// TIA Portal V19 export
FUNCTION "Area03_ITF" : Void   // FC22, LAD
// stored: SetENOAutomatically false
BEGIN

REGION Network 2: AREA ITF
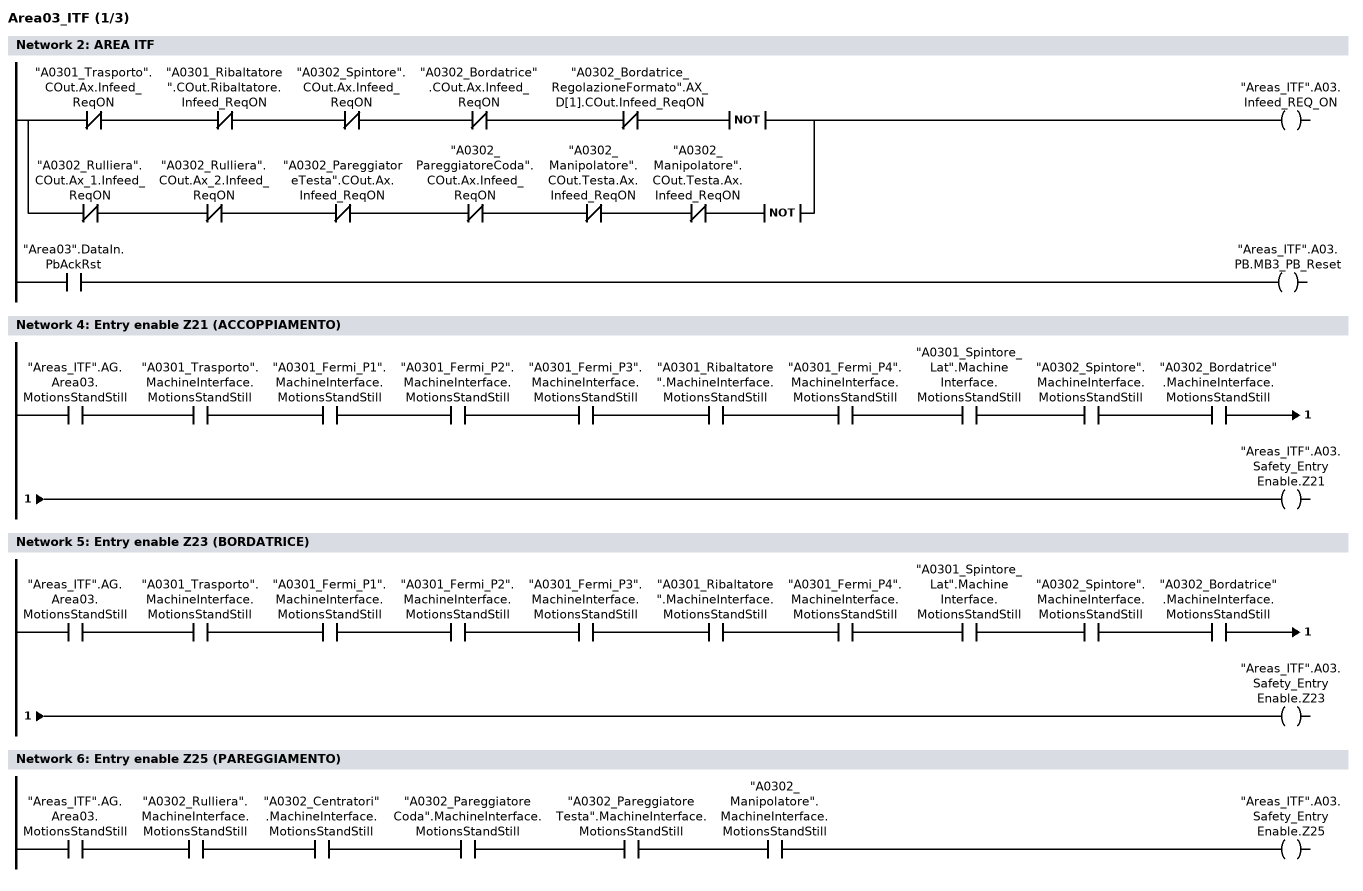
   RUNG wire#powerrail
      I_Contact( "A0301_Trasporto".COut.Ax.Infeed_ReqON )
      I_Contact( "A0301_Ribaltatore".COut.Ribaltatore.Infeed_ReqON )
      I_Contact( "A0302_Spintore".COut.Ax.Infeed_ReqON )
      I_Contact( "A0302_Bordatrice".COut.Ax.Infeed_ReqON )
      I_Contact( "A0302_Bordatrice_RegolazioneFormato".AX_D[1].COut.Infeed_ReqON )
      Not()
      wire#w1
      Coil( "Areas_ITF".A03.Infeed_REQ_ON )
   END_RUNG
   RUNG wire#powerrail
      I_Contact( "A0302_Rulliera".COut.Ax_1.Infeed_ReqON )
      I_Contact( "A0302_Rulliera".COut.Ax_2.Infeed_ReqON )
      I_Contact( "A0302_PareggiatoreTesta".COut.Ax.Infeed_ReqON )
      I_Contact( "A0302_PareggiatoreCoda".COut.Ax.Infeed_ReqON )
      I_Contact( "A0302_Manipolatore".COut.Testa.Ax.Infeed_ReqON )
      I_Contact( "A0302_Manipolatore".COut.Testa.Ax.Infeed_ReqON )
      Not()
   END_RUNG wire#w1
   RUNG wire#powerrail
      Contact( "Area03".DataIn.PbAckRst )
      Coil( "Areas_ITF".A03.PB.MB3_PB_Reset )
   END_RUNG
   // the same network as SCL:
   "Areas_ITF".A03.Infeed_REQ_ON := NOT (NOT "A0301_Trasporto".COut.Ax.Infeed_ReqON AND NOT "A0301_Ribaltatore".COut.Ribaltatore.Infeed_ReqON AND NOT "A0302_Spintore".COut.Ax.Infeed_ReqON AND NOT "A0302_Bordatrice".COut.Ax.Infeed_ReqON AND NOT "A0302_Bordatrice_RegolazioneFormato".AX_D[1].COut.Infeed_ReqON) OR NOT (NOT "A0302_Rulliera".COut.Ax_1.Infeed_ReqON AND NOT "A0302_Rulliera".COut.Ax_2.Infeed_ReqON AND NOT "A0302_PareggiatoreTesta".COut.Ax.Infeed_ReqON AND NOT "A0302_PareggiatoreCoda".COut.Ax.Infeed_ReqON AND NOT "A0302_Manipolatore".COut.Testa.Ax.Infeed_ReqON AND NOT "A0302_Manipolatore".COut.Testa.Ax.Infeed_ReqON);
   "Areas_ITF".A03.PB.MB3_PB_Reset := "Area03".DataIn.PbAckRst;
END_REGION

REGION Network 3: >
END_REGION

REGION Network 4: Entry enable Z21 (ACCOPPIAMENTO)
   RUNG wire#powerrail
      Contact( "Areas_ITF".AG.Area03.MotionsStandStill )
      Contact( "A0301_Trasporto".MachineInterface.MotionsStandStill )
      Contact( "A0301_Fermi_P1".MachineInterface.MotionsStandStill )
      Contact( "A0301_Fermi_P2".MachineInterface.MotionsStandStill )
      Contact( "A0301_Fermi_P3".MachineInterface.MotionsStandStill )
      Contact( "A0301_Ribaltatore".MachineInterface.MotionsStandStill )
      Contact( "A0301_Fermi_P4".MachineInterface.MotionsStandStill )
      Contact( "A0301_Spintore_Lat".MachineInterface.MotionsStandStill )
      Contact( "A0302_Spintore".MachineInterface.MotionsStandStill )
      Contact( "A0302_Bordatrice".MachineInterface.MotionsStandStill )
      Coil( "Areas_ITF".A03.Safety_EntryEnable.Z21 )
   END_RUNG
   // the same network as SCL:
   "Areas_ITF".A03.Safety_EntryEnable.Z21 := "Areas_ITF".AG.Area03.MotionsStandStill AND "A0301_Trasporto".MachineInterface.MotionsStandStill AND "A0301_Fermi_P1".MachineInterface.MotionsStandStill AND "A0301_Fermi_P2".MachineInterface.MotionsStandStill AND "A0301_Fermi_P3".MachineInterface.MotionsStandStill AND "A0301_Ribaltatore".MachineInterface.MotionsStandStill AND "A0301_Fermi_P4".MachineInterface.MotionsStandStill AND "A0301_Spintore_Lat".MachineInterface.MotionsStandStill AND "A0302_Spintore".MachineInterface.MotionsStandStill AND "A0302_Bordatrice".MachineInterface.MotionsStandStill;
END_REGION

REGION Network 5: Entry enable Z23 (BORDATRICE)
   RUNG wire#powerrail
      Contact( "Areas_ITF".AG.Area03.MotionsStandStill )
      Contact( "A0301_Trasporto".MachineInterface.MotionsStandStill )
      Contact( "A0301_Fermi_P1".MachineInterface.MotionsStandStill )
      Contact( "A0301_Fermi_P2".MachineInterface.MotionsStandStill )
      Contact( "A0301_Fermi_P3".MachineInterface.MotionsStandStill )
      Contact( "A0301_Ribaltatore".MachineInterface.MotionsStandStill )
      Contact( "A0301_Fermi_P4".MachineInterface.MotionsStandStill )
      Contact( "A0301_Spintore_Lat".MachineInterface.MotionsStandStill )
      Contact( "A0302_Spintore".MachineInterface.MotionsStandStill )
      Contact( "A0302_Bordatrice".MachineInterface.MotionsStandStill )
      Coil( "Areas_ITF".A03.Safety_EntryEnable.Z23 )
   END_RUNG
   // the same network as SCL:
   "Areas_ITF".A03.Safety_EntryEnable.Z23 := "Areas_ITF".AG.Area03.MotionsStandStill AND "A0301_Trasporto".MachineInterface.MotionsStandStill AND "A0301_Fermi_P1".MachineInterface.MotionsStandStill AND "A0301_Fermi_P2".MachineInterface.MotionsStandStill AND "A0301_Fermi_P3".MachineInterface.MotionsStandStill AND "A0301_Ribaltatore".MachineInterface.MotionsStandStill AND "A0301_Fermi_P4".MachineInterface.MotionsStandStill AND "A0301_Spintore_Lat".MachineInterface.MotionsStandStill AND "A0302_Spintore".MachineInterface.MotionsStandStill AND "A0302_Bordatrice".MachineInterface.MotionsStandStill;
END_REGION

REGION Network 6: Entry enable Z25 (PAREGGIAMENTO)
   RUNG wire#powerrail
      Contact( "Areas_ITF".AG.Area03.MotionsStandStill )
      Contact( "A0302_Rulliera".MachineInterface.MotionsStandStill )
      Contact( "A0302_Centratori".MachineInterface.MotionsStandStill )
      Contact( "A0302_PareggiatoreCoda".MachineInterface.MotionsStandStill )
      Contact( "A0302_PareggiatoreTesta".MachineInterface.MotionsStandStill )
      Contact( "A0302_Manipolatore".MachineInterface.MotionsStandStill )
      Coil( "Areas_ITF".A03.Safety_EntryEnable.Z25 )
   END_RUNG
   // the same network as SCL:
   "Areas_ITF".A03.Safety_EntryEnable.Z25 := "Areas_ITF".AG.Area03.MotionsStandStill AND "A0302_Rulliera".MachineInterface.MotionsStandStill AND "A0302_Centratori".MachineInterface.MotionsStandStill AND "A0302_PareggiatoreCoda".MachineInterface.MotionsStandStill AND "A0302_PareggiatoreTesta".MachineInterface.MotionsStandStill AND "A0302_Manipolatore".MachineInterface.MotionsStandStill;
END_REGION

REGION Network 7: < < < < CTRL SAFE > > > >
END_REGION

REGION Network 8: Ctrl Safe S120
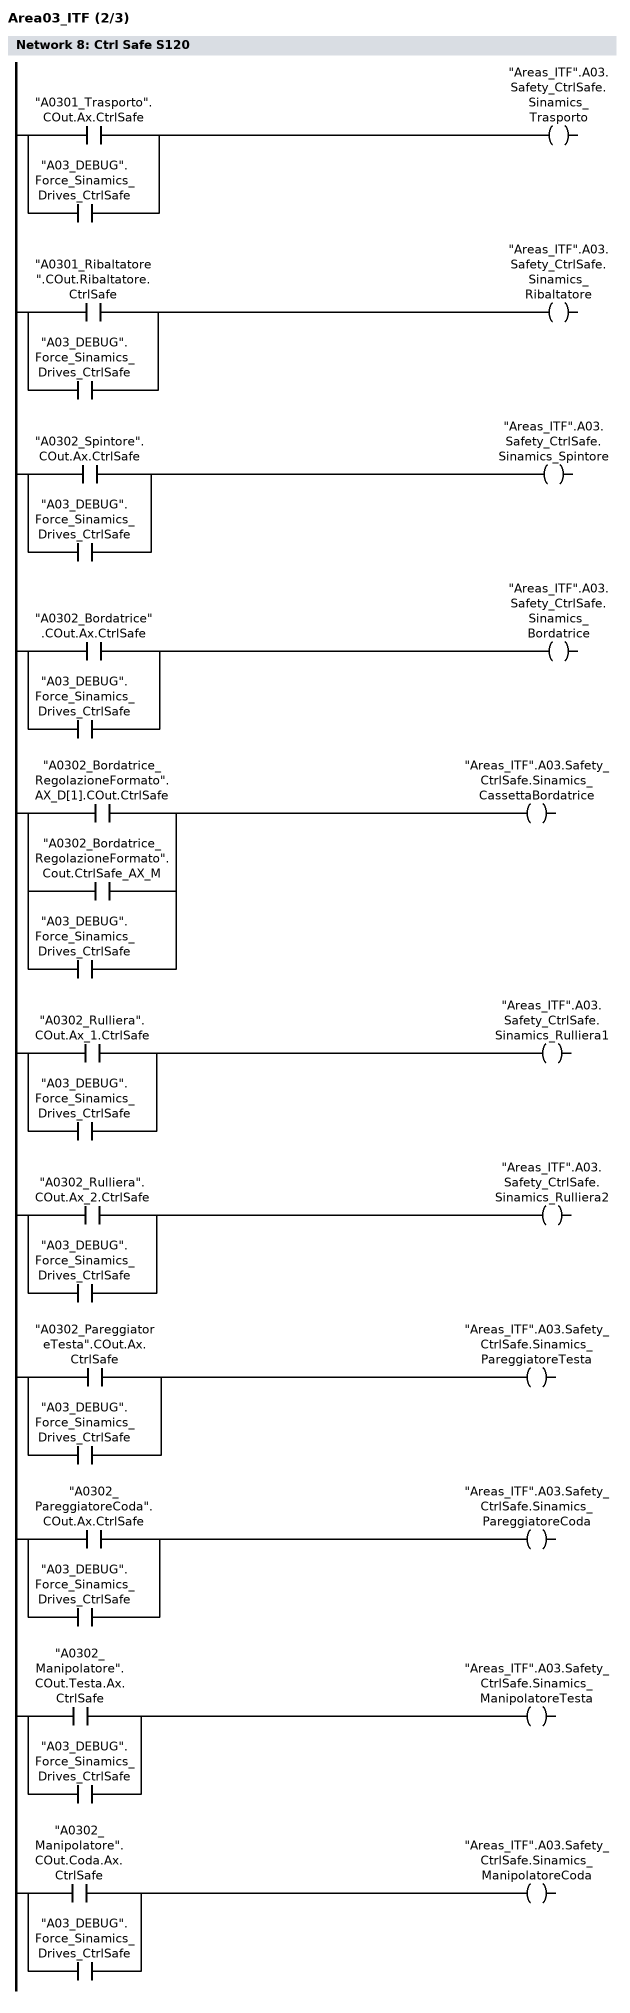
   RUNG wire#powerrail
      Contact( "A0301_Trasporto".COut.Ax.CtrlSafe )
      wire#w1
      Coil( "Areas_ITF".A03.Safety_CtrlSafe.Sinamics_Trasporto )
   END_RUNG
   RUNG wire#powerrail
      Contact( "A03_DEBUG".Force_Sinamics_Drives_CtrlSafe )
   END_RUNG wire#w1
   RUNG wire#powerrail
      Contact( "A0301_Ribaltatore".COut.Ribaltatore.CtrlSafe )
      wire#w2
      Coil( "Areas_ITF".A03.Safety_CtrlSafe.Sinamics_Ribaltatore )
   END_RUNG
   RUNG wire#powerrail
      Contact( "A03_DEBUG".Force_Sinamics_Drives_CtrlSafe )
   END_RUNG wire#w2
   RUNG wire#powerrail
      Contact( "A0302_Spintore".COut.Ax.CtrlSafe )
      wire#w3
      Coil( "Areas_ITF".A03.Safety_CtrlSafe.Sinamics_Spintore )
   END_RUNG
   RUNG wire#powerrail
      Contact( "A03_DEBUG".Force_Sinamics_Drives_CtrlSafe )
   END_RUNG wire#w3
   RUNG wire#powerrail
      Contact( "A0302_Bordatrice".COut.Ax.CtrlSafe )
      wire#w4
      Coil( "Areas_ITF".A03.Safety_CtrlSafe.Sinamics_Bordatrice )
   END_RUNG
   RUNG wire#powerrail
      Contact( "A03_DEBUG".Force_Sinamics_Drives_CtrlSafe )
   END_RUNG wire#w4
   RUNG wire#powerrail
      Contact( "A0302_Bordatrice_RegolazioneFormato".AX_D[1].COut.CtrlSafe )
      wire#w5
      Coil( "Areas_ITF".A03.Safety_CtrlSafe.Sinamics_CassettaBordatrice )
   END_RUNG
   RUNG wire#powerrail
      Contact( "A0302_Bordatrice_RegolazioneFormato".Cout.CtrlSafe_AX_M )
   END_RUNG wire#w5
   RUNG wire#powerrail
      Contact( "A03_DEBUG".Force_Sinamics_Drives_CtrlSafe )
   END_RUNG wire#w5
   RUNG wire#powerrail
      Contact( "A0302_Rulliera".COut.Ax_1.CtrlSafe )
      wire#w6
      Coil( "Areas_ITF".A03.Safety_CtrlSafe.Sinamics_Rulliera1 )
   END_RUNG
   RUNG wire#powerrail
      Contact( "A03_DEBUG".Force_Sinamics_Drives_CtrlSafe )
   END_RUNG wire#w6
   RUNG wire#powerrail
      Contact( "A0302_Rulliera".COut.Ax_2.CtrlSafe )
      wire#w7
      Coil( "Areas_ITF".A03.Safety_CtrlSafe.Sinamics_Rulliera2 )
   END_RUNG
   RUNG wire#powerrail
      Contact( "A03_DEBUG".Force_Sinamics_Drives_CtrlSafe )
   END_RUNG wire#w7
   RUNG wire#powerrail
      Contact( "A0302_PareggiatoreTesta".COut.Ax.CtrlSafe )
      wire#w8
      Coil( "Areas_ITF".A03.Safety_CtrlSafe.Sinamics_PareggiatoreTesta )
   END_RUNG
   RUNG wire#powerrail
      Contact( "A03_DEBUG".Force_Sinamics_Drives_CtrlSafe )
   END_RUNG wire#w8
   RUNG wire#powerrail
      Contact( "A0302_PareggiatoreCoda".COut.Ax.CtrlSafe )
      wire#w9
      Coil( "Areas_ITF".A03.Safety_CtrlSafe.Sinamics_PareggiatoreCoda )
   END_RUNG
   RUNG wire#powerrail
      Contact( "A03_DEBUG".Force_Sinamics_Drives_CtrlSafe )
   END_RUNG wire#w9
   RUNG wire#powerrail
      Contact( "A0302_Manipolatore".COut.Testa.Ax.CtrlSafe )
      wire#w10
      Coil( "Areas_ITF".A03.Safety_CtrlSafe.Sinamics_ManipolatoreTesta )
   END_RUNG
   RUNG wire#powerrail
      Contact( "A03_DEBUG".Force_Sinamics_Drives_CtrlSafe )
   END_RUNG wire#w10
   RUNG wire#powerrail
      Contact( "A0302_Manipolatore".COut.Coda.Ax.CtrlSafe )
      wire#w11
      Coil( "Areas_ITF".A03.Safety_CtrlSafe.Sinamics_ManipolatoreCoda )
   END_RUNG
   RUNG wire#powerrail
      Contact( "A03_DEBUG".Force_Sinamics_Drives_CtrlSafe )
   END_RUNG wire#w11
   // the same network as SCL:
   "Areas_ITF".A03.Safety_CtrlSafe.Sinamics_Trasporto := "A0301_Trasporto".COut.Ax.CtrlSafe OR "A03_DEBUG".Force_Sinamics_Drives_CtrlSafe;
   "Areas_ITF".A03.Safety_CtrlSafe.Sinamics_Ribaltatore := "A0301_Ribaltatore".COut.Ribaltatore.CtrlSafe OR "A03_DEBUG".Force_Sinamics_Drives_CtrlSafe;
   "Areas_ITF".A03.Safety_CtrlSafe.Sinamics_Spintore := "A0302_Spintore".COut.Ax.CtrlSafe OR "A03_DEBUG".Force_Sinamics_Drives_CtrlSafe;
   "Areas_ITF".A03.Safety_CtrlSafe.Sinamics_Bordatrice := "A0302_Bordatrice".COut.Ax.CtrlSafe OR "A03_DEBUG".Force_Sinamics_Drives_CtrlSafe;
   "Areas_ITF".A03.Safety_CtrlSafe.Sinamics_CassettaBordatrice := "A0302_Bordatrice_RegolazioneFormato".AX_D[1].COut.CtrlSafe OR "A0302_Bordatrice_RegolazioneFormato".Cout.CtrlSafe_AX_M OR "A03_DEBUG".Force_Sinamics_Drives_CtrlSafe;
   "Areas_ITF".A03.Safety_CtrlSafe.Sinamics_Rulliera1 := "A0302_Rulliera".COut.Ax_1.CtrlSafe OR "A03_DEBUG".Force_Sinamics_Drives_CtrlSafe;
   "Areas_ITF".A03.Safety_CtrlSafe.Sinamics_Rulliera2 := "A0302_Rulliera".COut.Ax_2.CtrlSafe OR "A03_DEBUG".Force_Sinamics_Drives_CtrlSafe;
   "Areas_ITF".A03.Safety_CtrlSafe.Sinamics_PareggiatoreTesta := "A0302_PareggiatoreTesta".COut.Ax.CtrlSafe OR "A03_DEBUG".Force_Sinamics_Drives_CtrlSafe;
   "Areas_ITF".A03.Safety_CtrlSafe.Sinamics_PareggiatoreCoda := "A0302_PareggiatoreCoda".COut.Ax.CtrlSafe OR "A03_DEBUG".Force_Sinamics_Drives_CtrlSafe;
   "Areas_ITF".A03.Safety_CtrlSafe.Sinamics_ManipolatoreTesta := "A0302_Manipolatore".COut.Testa.Ax.CtrlSafe OR "A03_DEBUG".Force_Sinamics_Drives_CtrlSafe;
   "Areas_ITF".A03.Safety_CtrlSafe.Sinamics_ManipolatoreCoda := "A0302_Manipolatore".COut.Coda.Ax.CtrlSafe OR "A03_DEBUG".Force_Sinamics_Drives_CtrlSafe;
END_REGION

REGION Network 9: Ctrl Safe Safety Valve
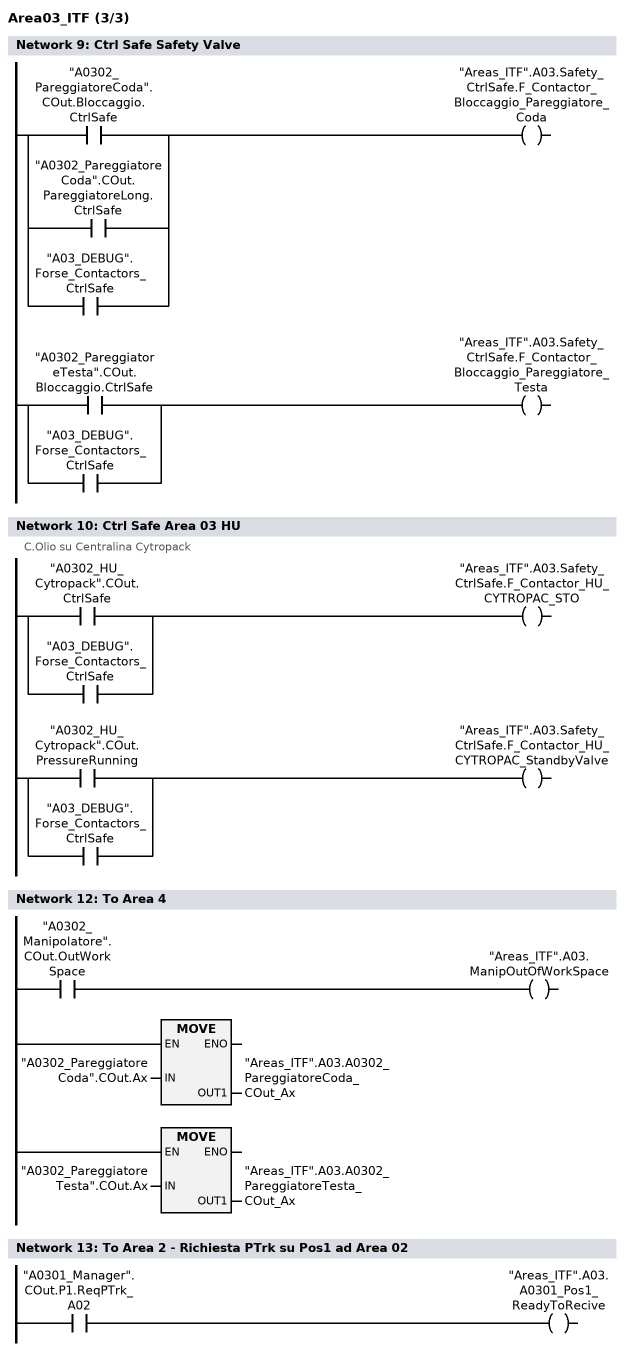
   RUNG wire#powerrail
      Contact( "A0302_PareggiatoreCoda".COut.Bloccaggio.CtrlSafe )
      wire#w1
      Coil( "Areas_ITF".A03.Safety_CtrlSafe.F_Contactor_Bloccaggio_Pareggiatore_Coda )
   END_RUNG
   RUNG wire#powerrail
      Contact( "A0302_PareggiatoreCoda".COut.PareggiatoreLong.CtrlSafe )
   END_RUNG wire#w1
   RUNG wire#powerrail
      Contact( "A03_DEBUG".Forse_Contactors_CtrlSafe )
   END_RUNG wire#w1
   RUNG wire#powerrail
      Contact( "A0302_PareggiatoreTesta".COut.Bloccaggio.CtrlSafe )
      wire#w2
      Coil( "Areas_ITF".A03.Safety_CtrlSafe.F_Contactor_Bloccaggio_Pareggiatore_Testa )
   END_RUNG
   RUNG wire#powerrail
      Contact( "A03_DEBUG".Forse_Contactors_CtrlSafe )
   END_RUNG wire#w2
   // the same network as SCL:
   "Areas_ITF".A03.Safety_CtrlSafe.F_Contactor_Bloccaggio_Pareggiatore_Coda := "A0302_PareggiatoreCoda".COut.Bloccaggio.CtrlSafe OR "A0302_PareggiatoreCoda".COut.PareggiatoreLong.CtrlSafe OR "A03_DEBUG".Forse_Contactors_CtrlSafe;
   "Areas_ITF".A03.Safety_CtrlSafe.F_Contactor_Bloccaggio_Pareggiatore_Testa := "A0302_PareggiatoreTesta".COut.Bloccaggio.CtrlSafe OR "A03_DEBUG".Forse_Contactors_CtrlSafe;
END_REGION

REGION Network 10: Ctrl Safe Area 03 HU
   // C.Olio su Centralina Cytropack
   RUNG wire#powerrail
      Contact( "A0302_HU_Cytropack".COut.CtrlSafe )
      wire#w1
      Coil( "Areas_ITF".A03.Safety_CtrlSafe.F_Contactor_HU_CYTROPAC_STO )
   END_RUNG
   RUNG wire#powerrail
      Contact( "A03_DEBUG".Forse_Contactors_CtrlSafe )
   END_RUNG wire#w1
   RUNG wire#powerrail
      Contact( "A0302_HU_Cytropack".COut.PressureRunning )
      wire#w2
      Coil( "Areas_ITF".A03.Safety_CtrlSafe.F_Contactor_HU_CYTROPAC_StandbyValve )
   END_RUNG
   RUNG wire#powerrail
      Contact( "A03_DEBUG".Forse_Contactors_CtrlSafe )
   END_RUNG wire#w2
   // the same network as SCL:
   "Areas_ITF".A03.Safety_CtrlSafe.F_Contactor_HU_CYTROPAC_STO := "A0302_HU_Cytropack".COut.CtrlSafe OR "A03_DEBUG".Forse_Contactors_CtrlSafe;
   "Areas_ITF".A03.Safety_CtrlSafe.F_Contactor_HU_CYTROPAC_StandbyValve := "A0302_HU_Cytropack".COut.PressureRunning OR "A03_DEBUG".Forse_Contactors_CtrlSafe;
END_REGION

REGION Network 12: To Area 4
   RUNG wire#powerrail
      Contact( "A0302_Manipolatore".COut.OutWorkSpace )
      Coil( "Areas_ITF".A03.ManipOutOfWorkSpace )
   END_RUNG
   RUNG wire#powerrail
      Move(in := "A0302_PareggiatoreCoda".COut.Ax, out1 => "Areas_ITF".A03.A0302_PareggiatoreCoda_COut_Ax)
   END_RUNG
   RUNG wire#powerrail
      Move(in := "A0302_PareggiatoreTesta".COut.Ax, out1 => "Areas_ITF".A03.A0302_PareggiatoreTesta_COut_Ax)
   END_RUNG
   // the same network as SCL:
   "Areas_ITF".A03.ManipOutOfWorkSpace := "A0302_Manipolatore".COut.OutWorkSpace;
   "Areas_ITF".A03.A0302_PareggiatoreCoda_COut_Ax := "A0302_PareggiatoreCoda".COut.Ax;
   "Areas_ITF".A03.A0302_PareggiatoreTesta_COut_Ax := "A0302_PareggiatoreTesta".COut.Ax;
END_REGION

REGION Network 13: To Area 2 - Richiesta PTrk su Pos1 ad Area 02
   RUNG wire#powerrail
      Contact( "A0301_Manager".COut.P1.ReqPTrk_A02 )
      Coil( "Areas_ITF".A03.A0301_Pos1_ReadyToRecive )
   END_RUNG
   // the same network as SCL:
   "Areas_ITF".A03.A0301_Pos1_ReadyToRecive := "A0301_Manager".COut.P1.ReqPTrk_A02;
END_REGION

REGION Network 14 (SCL): Area ITF Orchestrator
   // TRASFERIMENTO AREA INTERFACE SU ITF
   "Areas_ITF".A03.AreaInterface := "Area03".AreaInterface;


   "Areas_ITF".A03.Safety_SuperUser.PbSafetyReset := "A03_HMI".Area03.SuperUser.PbSafetyRst;
   "Areas_ITF".A03.Safety_SuperUser.SgnSafetyReset := "A03_HMI".Area03.SuperUser.SgnSafetyRst;

   "Areas_ITF".A03.Doors_Closed := NOT "F_DB".ZSI_Zone21.Door_NormalStop AND NOT "F_DB".ZSI_Zone23.Door_NormalStop AND NOT "F_DB".ZSI_Zone25.Door_NormalStop;
   "Areas_ITF".A03.Production_Running := "Sys".ByPass;

   //"Areas_ITF".A03.Production_Halted.Code :=;
   //"Areas_ITF".A03.Production_Halted.Message_N :=;

   "Areas_ITF".A03.SetUp_Bordatrice_Done := "A0302_Bordatrice_RegolazioneFormato".Cout.SetUp_Bordatrice_Done;

   //"MB3_Pb_Start_Ciclo_Area02" := "Areas_ITF".A02.PB.Area_DataOut_LampCycle;
   "Areas_ITF".A03.PB.MB3_Area02_PB_Start := FALSE;
   //"MB3_Pb_Start_Ciclo_Area02";
   "Areas_ITF".A03.PB.MB3_Area02_PB_Stop := FALSE;
   //"MB3_Pb_Stop_Ciclo_Area02";

   //"MB3_Pb_Start_Ciclo_Area01" := "Areas_ITF".A01.PB.Area_DataOut_LampCycle;
   "Areas_ITF".A03.PB.MB3_Area01_PB_Start := FALSE;
   //"MB3_Pb_Start_Ciclo_Area01";
   "Areas_ITF".A03.PB.MB3_Area01_PB_Stop := FALSE;
   //"MB3_Pb_Stop_Ciclo_Area01";
END_REGION
END_FUNCTION
